# EPICS substitutions: urRobotApp/Db/waypoints.substitutions
# Waypoints in joint space
file "$(URROBOT)/db/waypointJ.db"
{
pattern
{ N,              DESC,  J1,  J2,  J3,  J4,  J5,  J6,  SPEED,  ACCEL,  BLEND}
{ 1,  "WaypointJ $(N)",   0,   0,   0,   0,   0,   0,   0.50,   1.40,   0.00}
{ 2,  "WaypointJ $(N)",   0,   0,   0,   0,   0,   0,   0.50,   1.40,   0.00}
{ 3,  "WaypointJ $(N)",   0,   0,   0,   0,   0,   0,   0.50,   1.40,   0.00}
{ 4,  "WaypointJ $(N)",   0,   0,   0,   0,   0,   0,   0.50,   1.40,   0.00}
{ 5,  "WaypointJ $(N)",   0,   0,   0,   0,   0,   0,   0.50,   1.40,   0.00}
{ 6,  "WaypointJ $(N)",   0,   0,   0,   0,   0,   0,   0.50,   1.40,   0.00}
{ 7,  "WaypointJ $(N)",   0,   0,   0,   0,   0,   0,   0.50,   1.40,   0.00}
{ 8,  "WaypointJ $(N)",   0,   0,   0,   0,   0,   0,   0.50,   1.40,   0.00}
{ 9,  "WaypointJ $(N)",   0,   0,   0,   0,   0,   0,   0.50,   1.40,   0.00}
{10,  "WaypointJ $(N)",   0,   0,   0,   0,   0,   0,   0.50,   1.40,   0.00}
{11,  "WaypointJ $(N)",   0,   0,   0,   0,   0,   0,   0.50,   1.40,   0.00}
{12,  "WaypointJ $(N)",   0,   0,   0,   0,   0,   0,   0.50,   1.40,   0.00}
{13,  "WaypointJ $(N)",   0,   0,   0,   0,   0,   0,   0.50,   1.40,   0.00}
{14,  "WaypointJ $(N)",   0,   0,   0,   0,   0,   0,   0.50,   1.40,   0.00}
{15,  "WaypointJ $(N)",   0,   0,   0,   0,   0,   0,   0.50,   1.40,   0.00}
{16,  "WaypointJ $(N)",   0,   0,   0,   0,   0,   0,   0.50,   1.40,   0.00}
{17,  "WaypointJ $(N)",   0,   0,   0,   0,   0,   0,   0.50,   1.40,   0.00}
{18,  "WaypointJ $(N)",   0,   0,   0,   0,   0,   0,   0.50,   1.40,   0.00}
{19,  "WaypointJ $(N)",   0,   0,   0,   0,   0,   0,   0.50,   1.40,   0.00}
{20,  "WaypointJ $(N)",   0,   0,   0,   0,   0,   0,   0.50,   1.40,   0.00}
{21,  "WaypointJ $(N)",   0,   0,   0,   0,   0,   0,   0.50,   1.40,   0.00}
{22,  "WaypointJ $(N)",   0,   0,   0,   0,   0,   0,   0.50,   1.40,   0.00}
{23,  "WaypointJ $(N)",   0,   0,   0,   0,   0,   0,   0.50,   1.40,   0.00}
{24,  "WaypointJ $(N)",   0,   0,   0,   0,   0,   0,   0.50,   1.40,   0.00}
{25,  "WaypointJ $(N)",   0,   0,   0,   0,   0,   0,   0.50,   1.40,   0.00}
{26,  "WaypointJ $(N)",   0,   0,   0,   0,   0,   0,   0.50,   1.40,   0.00}
{27,  "WaypointJ $(N)",   0,   0,   0,   0,   0,   0,   0.50,   1.40,   0.00}
{28,  "WaypointJ $(N)",   0,   0,   0,   0,   0,   0,   0.50,   1.40,   0.00}
{29,  "WaypointJ $(N)",   0,   0,   0,   0,   0,   0,   0.50,   1.40,   0.00}
{30,  "WaypointJ $(N)",   0,   0,   0,   0,   0,   0,   0.50,   1.40,   0.00}
}

# Waypoints in Cartesian space
file "$(URROBOT)/db/waypointL.db"
{
pattern
{ N,              DESC,  X,  Y,  Z,  ROLL,  PITCH,  YAW,  SPEED,  ACCEL,  BLEND}
{ 1,  "WaypointL $(N)",  0,  0,  0,     0,      0,    0,   0.50,   1.40,   0.00}
{ 2,  "WaypointL $(N)",  0,  0,  0,     0,      0,    0,   0.50,   1.40,   0.00}
{ 3,  "WaypointL $(N)",  0,  0,  0,     0,      0,    0,   0.50,   1.40,   0.00}
{ 4,  "WaypointL $(N)",  0,  0,  0,     0,      0,    0,   0.50,   1.40,   0.00}
{ 5,  "WaypointL $(N)",  0,  0,  0,     0,      0,    0,   0.50,   1.40,   0.00}
{ 6,  "WaypointL $(N)",  0,  0,  0,     0,      0,    0,   0.50,   1.40,   0.00}
{ 7,  "WaypointL $(N)",  0,  0,  0,     0,      0,    0,   0.50,   1.40,   0.00}
{ 8,  "WaypointL $(N)",  0,  0,  0,     0,      0,    0,   0.50,   1.40,   0.00}
{ 9,  "WaypointL $(N)",  0,  0,  0,     0,      0,    0,   0.50,   1.40,   0.00}
{10,  "WaypointL $(N)",  0,  0,  0,     0,      0,    0,   0.50,   1.40,   0.00}
{11,  "WaypointL $(N)",  0,  0,  0,     0,      0,    0,   0.50,   1.40,   0.00}
{12,  "WaypointL $(N)",  0,  0,  0,     0,      0,    0,   0.50,   1.40,   0.00}
{13,  "WaypointL $(N)",  0,  0,  0,     0,      0,    0,   0.50,   1.40,   0.00}
{14,  "WaypointL $(N)",  0,  0,  0,     0,      0,    0,   0.50,   1.40,   0.00}
{15,  "WaypointL $(N)",  0,  0,  0,     0,      0,    0,   0.50,   1.40,   0.00}
{16,  "WaypointL $(N)",  0,  0,  0,     0,      0,    0,   0.50,   1.40,   0.00}
{17,  "WaypointL $(N)",  0,  0,  0,     0,      0,    0,   0.50,   1.40,   0.00}
{18,  "WaypointL $(N)",  0,  0,  0,     0,      0,    0,   0.50,   1.40,   0.00}
{19,  "WaypointL $(N)",  0,  0,  0,     0,      0,    0,   0.50,   1.40,   0.00}
{20,  "WaypointL $(N)",  0,  0,  0,     0,      0,    0,   0.50,   1.40,   0.00}
{21,  "WaypointL $(N)",  0,  0,  0,     0,      0,    0,   0.50,   1.40,   0.00}
{22,  "WaypointL $(N)",  0,  0,  0,     0,      0,    0,   0.50,   1.40,   0.00}
{23,  "WaypointL $(N)",  0,  0,  0,     0,      0,    0,   0.50,   1.40,   0.00}
{24,  "WaypointL $(N)",  0,  0,  0,     0,      0,    0,   0.50,   1.40,   0.00}
{25,  "WaypointL $(N)",  0,  0,  0,     0,      0,    0,   0.50,   1.40,   0.00}
{26,  "WaypointL $(N)",  0,  0,  0,     0,      0,    0,   0.50,   1.40,   0.00}
{27,  "WaypointL $(N)",  0,  0,  0,     0,      0,    0,   0.50,   1.40,   0.00}
{28,  "WaypointL $(N)",  0,  0,  0,     0,      0,    0,   0.50,   1.40,   0.00}
{29,  "WaypointL $(N)",  0,  0,  0,     0,      0,    0,   0.50,   1.40,   0.00}
{30,  "WaypointL $(N)",  0,  0,  0,     0,      0,    0,   0.50,   1.40,   0.00}
}

# 10 waypoint actions
file "$(URROBOT)/db/waypoint_actions10.db" {{}}
